# B&R Automation Studio project AS_Target_Simulink_Test (part 6)

#### sltestCruiseControlDefective.h
```c
/********************************************************************
 * COPYRIGHT -- Bernecker + Rainer Industrie-Elektronik Ges.m.b.H.
 ********************************************************************
 * Program: sltestCruiseControlDefective
 * File: sltestCruiseControlDefective.h
 * Author: The MathWorks, Inc.
 * Created: Wed Aug 30 21:41:02 2006
 ********************************************************************
 * Header for program sltestCruiseControlDefective
 ********************************************************************
 * Generated with B&R Automation Studio Target for Simulink  V6.1.0
 * (ERT based)
 ********************************************************************/

#ifndef RTW_HEADER_sltestCruiseControlDefective_h_
#define RTW_HEADER_sltestCruiseControlDefective_h_
#include <math.h>
#ifndef sltestCruiseControlDefective_COMMON_INCLUDES_
# define sltestCruiseControlDefective_COMMON_INCLUDES_
#include "rtwtypes.h"
#include "rtw_continuous.h"
#include "rtw_solver.h"
#endif                       /* sltestCruiseControlDefective_COMMON_INCLUDES_ */

#include <bur/plctypes.h>

#ifdef _DEFAULT_INCLUDES
 #include <AsDefault.h>
#endif

#ifndef AST_ROUND
#define AST_ROUND(x) ((x)>=0?(long long)((x)+0.5):(long long)((x)-0.5))
#endif

#include "sltestCruiseControlDefective_types.h"

/* Macros for accessing real-time model data structure */
#ifndef rtmGetErrorStatus
# define rtmGetErrorStatus(rtm)        ((rtm)->errorStatus)
#endif

#ifndef rtmSetErrorStatus
# define rtmSetErrorStatus(rtm, val)   ((rtm)->errorStatus = (val))
#endif

#ifndef rtmGetT
# define rtmGetT(rtm)                  (rtmGetTPtr((rtm))[0])
#endif

#ifndef rtmGetTPtr
# define rtmGetTPtr(rtm)               ((rtm)->Timing.t)
#endif

#ifndef MIN
#define MIN(a,b)                       ((a) < (b) ? (a) : (b))
#endif

#ifndef MAX
#define MAX(a,b)                       ((a) > (b) ? (a) : (b))
#endif

/* Block signals (default storage) */
typedef struct {
  real_T Sum1;                         /* '<S1>/Sum1' */
  boolean_T ActiveControl;             /* '<S1>/Logical Operator' */
} BlockIO_sltestCruiseControlDefe;

/* Block states (default storage) for system '<Root>' */
typedef struct {
  real_T UnitDelay_DSTATE;             /* '<S1>/Unit Delay' */
  real_T DiscreteTimeIntegrator_DSTATE;/* '<S5>/Discrete-Time Integrator' */
  struct {
    void *TimePtr;
    void *DataPtr;
    void *RSimInfoPtr;
  } FromWs_PWORK;                      /* '<S2>/FromWs' */

  struct {
    int_T PrevIndex;
  } FromWs_IWORK;                      /* '<S2>/FromWs' */

  boolean_T UnitDelay1_DSTATE;         /* '<S1>/Unit Delay1' */
} D_Work_sltestCruiseControlDefec;

/* External outputs (root outports fed by signals with default storage) */
typedef struct {
  real_T throt;                        /* '<Root>/throt' */
  real_T target;                       /* '<Root>/target' */
} ExternalOutputs_sltestCruiseCon;

/* Parameters (default storage) */
struct Parameters_sltestCruiseControlD_ {
  real_T Constant3_Value;              /* Expression: 1
                                        * Referenced by: '<S1>/Constant3'
                                        */
  real_T Constant1_Value;              /* Expression: 1
                                        * Referenced by: '<S1>/Constant1'
                                        */
  real_T throt_Y0;                     /* Expression: 0
                                        * Referenced by: '<S5>/throt'
                                        */
  real_T DiscreteTimeIntegrator_gainval;
                           /* Computed Parameter: DiscreteTimeIntegrator_gainval
                            * Referenced by: '<S5>/Discrete-Time Integrator'
                            */
  real_T DiscreteTimeIntegrator_IC;    /* Expression: 0
                                        * Referenced by: '<S5>/Discrete-Time Integrator'
                                        */
  real_T DiscreteTimeIntegrator_UpperSat;/* Expression: 5
                                          * Referenced by: '<S5>/Discrete-Time Integrator'
                                          */
  real_T DiscreteTimeIntegrator_LowerSat;/* Expression: -5
                                          * Referenced by: '<S5>/Discrete-Time Integrator'
                                          */
  real_T Kp1_Gain;                     /* Expression: 0.01
                                        * Referenced by: '<S5>/Kp1'
                                        */
  real_T Kp_Gain;                      /* Expression: 0.02
                                        * Referenced by: '<S5>/Kp'
                                        */
  real_T UnitDelay_InitialCondition;   /* Expression: 0
                                        * Referenced by: '<S1>/Unit Delay'
                                        */
  boolean_T UnitDelay1_InitialCondition;
                              /* Computed Parameter: UnitDelay1_InitialCondition
                               * Referenced by: '<S1>/Unit Delay1'
                               */
};

/* Real-time Model Data Structure */
struct tag_RTM_sltestCruiseControlDefe {
  const char_T *errorStatus;
  RTWSolverInfo solverInfo;

  /*
   * Timing:
   * The following substructure contains information regarding
   * the timing information for the model.
   */
  struct {
    uint32_T clockTick0;
    uint32_T clockTickH0;
    time_T stepSize0;
    uint32_T clockTick1;
    uint32_T clockTickH1;
    SimTimeStep simTimeStep;
    time_T *t;
    time_T tArray[2];
  } Timing;
};

/* Block parameters (default storage) */
extern Parameters_sltestCruiseControlD sltestCruiseControlDefective_P;

/* Block signals (default storage) */
extern BlockIO_sltestCruiseControlDefe sltestCruiseControlDefective_B;

/* Block states (default storage) */
extern D_Work_sltestCruiseControlDefec sltestCruiseControlDefect_DWork;

/* External outputs (root outports fed by signals with default storage) */
extern ExternalOutputs_sltestCruiseCon sltestCruiseControlDefective_Y;

/* Model entry point functions */
extern void sltestCruiseControlDefective_initialize(void);
extern void sltestCruiseControlDefective_output(void);
extern void sltestCruiseControlDefective_update(void);
extern void sltestCruiseControlDefective_terminate(void);

/* Real-time Model object */
extern RT_MODEL_sltestCruiseControlDef *const sltestCruiseControlDefective_M;

/*-
 * The generated code includes comments that allow you to trace directly
 * back to the appropriate location in the model.  The basic format
 * is <system>/block_name, where system is the system number (uniquely
 * assigned by Simulink) and block_name is the name of the block.
 *
 * Use the MATLAB hilite_system command to trace the generated code back
 * to the model.  For example,
 *
 * hilite_system('<S3>')    - opens system 3
 * hilite_system('<S3>/Kp') - opens and selects block Kp which resides in S3
 *
 * Here is the system hierarchy for this model
 *
 * '<Root>' : 'sltestCruiseControlDefective'
 * '<S1>'   : 'sltestCruiseControlDefective/Controller'
 * '<S2>'   : 'sltestCruiseControlDefective/Inputs'
 * '<S3>'   : 'sltestCruiseControlDefective/Safety Properties'
 * '<S4>'   : 'sltestCruiseControlDefective/Size-Type'
 * '<S5>'   : 'sltestCruiseControlDefective/Controller/PI Controller'
 * '<S6>'   : 'sltestCruiseControlDefective/Safety Properties/Implies'
 * '<S7>'   : 'sltestCruiseControlDefective/Safety Properties/constraint'
 * '<S8>'   : 'sltestCruiseControlDefective/Safety Properties/constraint/viewdvc'
 * '<S9>'   : 'sltestCruiseControlDefective/Size-Type/Bus1'
 */
#endif                          /* RTW_HEADER_sltestCruiseControlDefective_h_ */
```

#### sltestCruiseControlDefective_data.c
```c
/********************************************************************
 * COPYRIGHT -- Bernecker + Rainer Industrie-Elektronik Ges.m.b.H.
 ********************************************************************
 * Program: sltestCruiseControlDefective
 * File: sltestCruiseControlDefective_data.c
 * Author: The MathWorks, Inc.
 * Created: Wed Aug 30 21:41:02 2006
 ********************************************************************
 * Data for program sltestCruiseControlDefective
 ********************************************************************
 * Generated with B&R Automation Studio Target for Simulink  V6.1.0
 * (ERT based)
 ********************************************************************/

#include "sltestCruiseControlDefective.h"
#include "sltestCruiseControlDefective_private.h"

/*  GLOBAL DATA DEFINITIONS */

/* Block parameters (default storage) */
Parameters_sltestCruiseControlD sltestCruiseControlDefective_P = {
  /* Expression: 1
   * Referenced by: '<S1>/Constant3'
   */
  1.0,

  /* Expression: 1
   * Referenced by: '<S1>/Constant1'
   */
  1.0,

  /* Expression: 0
   * Referenced by: '<S5>/throt'
   */
  0.0,

  /* Computed Parameter: DiscreteTimeIntegrator_gainval
   * Referenced by: '<S5>/Discrete-Time Integrator'
   */
  0.01,

  /* Expression: 0
   * Referenced by: '<S5>/Discrete-Time Integrator'
   */
  0.0,

  /* Expression: 5
   * Referenced by: '<S5>/Discrete-Time Integrator'
   */
  5.0,

  /* Expression: -5
   * Referenced by: '<S5>/Discrete-Time Integrator'
   */
  -5.0,

  /* Expression: 0.01
   * Referenced by: '<S5>/Kp1'
   */
  0.01,

  /* Expression: 0.02
   * Referenced by: '<S5>/Kp'
   */
  0.02,

  /* Expression: 0
   * Referenced by: '<S1>/Unit Delay'
   */
  0.0,

  /* Computed Parameter: UnitDelay1_InitialCondition
   * Referenced by: '<S1>/Unit Delay1'
   */
  0
};
```

#### sltestCruiseControlDefective_private.h
```c
/********************************************************************
 * COPYRIGHT -- Bernecker + Rainer Industrie-Elektronik Ges.m.b.H.
 ********************************************************************
 * Program: sltestCruiseControlDefective
 * File: sltestCruiseControlDefective_private.h
 * Author: The MathWorks, Inc.
 * Created: Wed Aug 30 21:41:02 2006
 ********************************************************************
 * Header for program sltestCruiseControlDefective
 ********************************************************************
 * Generated with B&R Automation Studio Target for Simulink  V6.1.0
 * (ERT based)
 ********************************************************************/

#ifndef RTW_HEADER_sltestCruiseControlDefective_private_h_
#define RTW_HEADER_sltestCruiseControlDefective_private_h_
#include "rtwtypes.h"
#define _ASMATH_
#define ASMATH_
#define _ASMATH_H
#define ASMATH_H
#define _ASMATH_H_
#define ASMATH_H_
#define _ASSTRING_
#define ASSTRING_
#define _ASSTRING_H
#define ASSTRING_H
#define _ASSTRING_H_
#define ASSTRING_H_
#include <bur/plctypes.h>
#ifdef _DEFAULT_INCLUDES
#include <AsDefault.h>
#endif

/* Private macros used by the generated code to access rtModel */
#ifndef rtmIsMajorTimeStep
# define rtmIsMajorTimeStep(rtm)       (((rtm)->Timing.simTimeStep) == MAJOR_TIME_STEP)
#endif

#ifndef rtmIsMinorTimeStep
# define rtmIsMinorTimeStep(rtm)       (((rtm)->Timing.simTimeStep) == MINOR_TIME_STEP)
#endif

#ifndef rtmSetTPtr
# define rtmSetTPtr(rtm, val)          ((rtm)->Timing.t = (val))
#endif

/* Used by FromWorkspace Block: '<S2>/FromWs' */
#ifndef rtInterpolate
# define rtInterpolate(v1,v2,f1,f2)    (((v1)==(v2))?((double)(v1)): (((f1)*((double)(v1)))+((f2)*((double)(v2)))))
#endif

#ifndef rtRound
# define rtRound(v)                    ( ((v) >= 0) ? floor((v) + 0.5) : ceil((v) - 0.5) )
#endif

#ifndef MIN
#define MIN(a,b)                       ((a) < (b) ? (a) : (b))
#endif

#ifndef MAX
#define MAX(a,b)                       ((a) > (b) ? (a) : (b))
#endif
#endif                  /* RTW_HEADER_sltestCruiseControlDefective_private_h_ */
```

#### sltestCruiseControlDefective_types.h
```c
/********************************************************************
 * COPYRIGHT -- Bernecker + Rainer Industrie-Elektronik Ges.m.b.H.
 ********************************************************************
 * Program: sltestCruiseControlDefective
 * File: sltestCruiseControlDefective_types.h
 * Author: The MathWorks, Inc.
 * Created: Wed Aug 30 21:41:02 2006
 ********************************************************************
 * Header for program sltestCruiseControlDefective
 ********************************************************************
 * Generated with B&R Automation Studio Target for Simulink  V6.1.0
 * (ERT based)
 ********************************************************************/

#ifndef RTW_HEADER_sltestCruiseControlDefective_types_h_
#define RTW_HEADER_sltestCruiseControlDefective_types_h_
#include "rtwtypes.h"
#ifndef MIN
#define MIN(a,b)                       ((a) < (b) ? (a) : (b))
#endif

#ifndef MAX
#define MAX(a,b)                       ((a) > (b) ? (a) : (b))
#endif

#ifndef DEFINED_TYPEDEF_FOR_setpoint_
#define DEFINED_TYPEDEF_FOR_setpoint_

typedef struct {
  boolean_T inc;
  boolean_T dec;
} setpoint;

#endif

#ifndef DEFINED_TYPEDEF_FOR_Switches_
#define DEFINED_TYPEDEF_FOR_Switches_

typedef struct {
  boolean_T enable;
  boolean_T brake;
  boolean_T set;
  setpoint setIncDec;
} Switches;

#endif

#ifndef DEFINED_TYPEDEF_FOR_InputBus_
#define DEFINED_TYPEDEF_FOR_InputBus_

typedef struct {
  real_T Actual_speed;
  Switches Switches;
} InputBus;

#endif

/* Parameters (default storage) */
typedef struct Parameters_sltestCruiseControlD_ Parameters_sltestCruiseControlD;

/* Forward declaration for rtModel */
typedef struct tag_RTM_sltestCruiseControlDefe RT_MODEL_sltestCruiseControlDef;

#endif                    /* RTW_HEADER_sltestCruiseControlDefective_types_h_ */
```

#### task_properties.txt
```
For manual assignment to hardware configuration please
add the following additional include directories:

\Logical\MATLAB_includes\R2019b\

And the following additional build options:

-lm -D MODEL=sltestCruiseControlDefective -D NUMST=2 -D NCSTATES=0 -D HAVESTDIO -D MODEL_HAS_DYNAMICALLY_LOADED_SFCNS=0 -D CLASSIC_INTERFACE=0 -D ALLOCATIONFCN=0 -D TID01EQ=1 -D TERMFCN=1 -D ONESTEPFCN=0 -D MAT_FILE=0 -D MULTI_INSTANCE_CODE=0 -D INTEGER_CODE=0 -D MT=0
```

Listed in the project but not available here: Logical/MATLAB_includes/R2019b/MatlabEngine.hpp, Logical/MATLAB_includes/R2019b/bio_sig.h, Logical/MATLAB_includes/R2019b/blas.h, Logical/MATLAB_includes/R2019b/blascompat32.h, Logical/MATLAB_includes/R2019b/cg_matrx.h, Logical/MATLAB_includes/R2019b/cg_sfun.h, Logical/MATLAB_includes/R2019b/cgxert.h, Logical/MATLAB_includes/R2019b/dt_info.h, Logical/MATLAB_includes/R2019b/emlrt.h, Logical/MATLAB_includes/R2019b/engine.h, Logical/MATLAB_includes/R2019b/ext_share.h, Logical/MATLAB_includes/R2019b/ext_svr.h, Logical/MATLAB_includes/R2019b/ext_svr_transport.h, Logical/MATLAB_includes/R2019b/ext_test.h, Logical/MATLAB_includes/R2019b/ext_types.h, Logical/MATLAB_includes/R2019b/ext_work.h, Logical/MATLAB_includes/R2019b/fintrf.h, Logical/MATLAB_includes/R2019b/fixedpoint.h, Logical/MATLAB_includes/R2019b/fixpoint_spec.h, Logical/MATLAB_includes/R2019b/io64.h, Logical/MATLAB_includes/R2019b/lapack.h, Logical/MATLAB_includes/R2019b/lapacke.h, Logical/MATLAB_includes/R2019b/lapacke_config.h, Logical/MATLAB_includes/R2019b/libmwjpegreader.h, Logical/MATLAB_includes/R2019b/libmwrgb2gray_tbb.h, Logical/MATLAB_includes/R2019b/libmwrgb2hsv_tbb.h, Logical/MATLAB_includes/R2019b/mat.h, Logical/MATLAB_includes/R2019b/matrix.h, Logical/MATLAB_includes/R2019b/mdl_info.h, Logical/MATLAB_includes/R2019b/mem_mgr.h, Logical/MATLAB_includes/R2019b/mex.h, Logical/MATLAB_includes/R2019b/mwmathutil.h, Logical/MATLAB_includes/R2019b/odesup.h, Logical/MATLAB_includes/R2019b/polygonBoolean.h, Logical/MATLAB_includes/R2019b/pt_info.h, Logical/MATLAB_includes/R2019b/rt_logging.h, Logical/MATLAB_includes/R2019b/rt_logging_mmi.h, Logical/MATLAB_includes/R2019b/rt_math.h, Logical/MATLAB_includes/R2019b/rt_matrx.h, Logical/MATLAB_includes/R2019b/rt_mxclassid.h, Logical/MATLAB_includes/R2019b/rt_sim.h, Logical/MATLAB_includes/R2019b/rtiostream.h, Logical/MATLAB_includes/R2019b/rtmcmacros.h, Logical/MATLAB_includes/R2019b/rtmmacros.h, Logical/MATLAB_includes/R2019b/rtsplntypes.h, Logical/MATLAB_includes/R2019b/rtw_capi.h, Logical/MATLAB_includes/R2019b/rtw_capi_examples.h, Logical/MATLAB_includes/R2019b/rtw_continuous.h, Logical/MATLAB_includes/R2019b/rtw_extmode.h, Logical/MATLAB_includes/R2019b/rtw_linux.h, Logical/MATLAB_includes/R2019b/rtw_linux_mac.h, Logical/MATLAB_includes/R2019b/rtw_matlogging.h, Logical/MATLAB_includes/R2019b/rtw_modelmap.h, Logical/MATLAB_includes/R2019b/rtw_modelmap_logging.h, Logical/MATLAB_includes/R2019b/rtw_msvc_lshift.h, Logical/MATLAB_includes/R2019b/rtw_solver.h, Logical/MATLAB_includes/R2019b/rtw_windows.h, Logical/MATLAB_includes/R2019b/sfcn_bridge.h, Logical/MATLAB_includes/R2019b/sfcn_loader_c_api.h, Logical/MATLAB_includes/R2019b/sfun_rtwcg.hpp, Logical/MATLAB_includes/R2019b/sigmapdef_sfcn.h, Logical/MATLAB_includes/R2019b/sigregdef.h, Logical/MATLAB_includes/R2019b/sigstream_rtw.h, Logical/MATLAB_includes/R2019b/simlogCIntrf.h, Logical/MATLAB_includes/R2019b/simstruc.h, Logical/MATLAB_includes/R2019b/simstruc_compcond.h, Logical/MATLAB_includes/R2019b/simstruc_debug.h, Logical/MATLAB_includes/R2019b/simstruc_def.h, Logical/MATLAB_includes/R2019b/simstruc_internal.h, Logical/MATLAB_includes/R2019b/simstruc_types.h, Logical/MATLAB_includes/R2019b/simulink.h, Logical/MATLAB_includes/R2019b/simulink2.h, Logical/MATLAB_includes/R2019b/simulink_solver_api.h, Logical/MATLAB_includes/R2019b/sl_common_types_def.h, Logical/MATLAB_includes/R2019b/sl_datatype_access.h, Logical/MATLAB_includes/R2019b/sl_fileio_rtw.h, Logical/MATLAB_includes/R2019b/sl_fixpt.h, Logical/MATLAB_includes/R2019b/sl_prodhwdevicetype.h, Logical/MATLAB_includes/R2019b/sl_report_types.h, Logical/MATLAB_includes/R2019b/sl_sample_time_defs.h, Logical/MATLAB_includes/R2019b/sl_sfcn_st_api.h, Logical/MATLAB_includes/R2019b/sl_solver_rtw.h, Logical/MATLAB_includes/R2019b/sl_types_def.h, Logical/MATLAB_includes/R2019b/slexec_parallel.h, Logical/MATLAB_includes/R2019b/slexec_simbridge.h, Logical/MATLAB_includes/R2019b/slexec_simstruct_bridge.h, Logical/MATLAB_includes/R2019b/slexec_vm_lookup_functions.h, Logical/MATLAB_includes/R2019b/slexec_vm_rt_functions.h, Logical/MATLAB_includes/R2019b/slexec_vm_zc_functions.h, Logical/MATLAB_includes/R2019b/slsv_diagnostic_logger_type.h, Logical/MATLAB_includes/R2019b/slsv_mexhelper.h, Logical/MATLAB_includes/R2019b/solver_zc.h, Logical/MATLAB_includes/R2019b/sysran_types.h, Logical/MATLAB_includes/R2019b/updown.h, Logical/MATLAB_includes/R2019b/updown_util.h, Logical/MATLAB_includes/R2019b/upsup_public.h, Logical/MATLAB_includes/R2019b/sf_runtime/sf_runtime_spec.h, Logical/MATLAB_includes/R2019b/sf_runtime/sf_runtime_types.h, Logical/MATLAB_includes/R2019b/sf_runtime/sf_test_language.h, Logical/MATLAB_includes/R2019b/sf_runtime/sfc_api.h, Logical/MATLAB_includes/R2019b/sf_runtime/sfc_messages.h, Logical/MATLAB_includes/R2019b/sf_runtime/sfc_mex.h, Logical/MATLAB_includes/R2019b/sf_runtime/sfc_sf.h, Logical/MATLAB_includes/R2019b/sf_runtime/sfcdebug.h, Logical/MATLAB_includes/R2019b/sf_runtime/slTestResult.h, Logical/MATLAB_includes/R2019b/sf_runtime/slTestTypes.h, Logical/MATLAB_includes/R2019b/sf_runtime/utils.h, Logical/MATLAB_includes/R2019b/sf_runtime/ChartInfoStruct.h, Logical/Model/pend_mod/local.typ, Logical/Model/pend_mod/local.var, Logical/Controller/pend_ctrl/local.typ, Logical/TD_Test/local.typ, Logical/TD_Test/local.var, Logical/sltest/local.typ
